GLOBALCONSTANTS DefaultPool_Numeric (* Numeric object pool constants (ID, Scale, Offset, Decimals) *)
  PACKAGE Uebungen::const::UT;
  VAR_GLOBAL CONSTANT
    InputNumber_I3 : logiBUS::utils::conversion::phys::NumericObjectPool_S := (u16ObjId := 9002, r32Scale := 0.01, i32Offset := -100000, u8Decimals := 2);
    InputNumber_I4 : logiBUS::utils::conversion::phys::NumericObjectPool_S := (u16ObjId := 9003, r32Scale := 0.01, i32Offset := -100000, u8Decimals := 2);
    OutputNumber_N3 : logiBUS::utils::conversion::phys::NumericObjectPool_S := (u16ObjId := 12002, r32Scale := 0.01, i32Offset := -100000, u8Decimals := 2);
  END_VAR
END_GLOBALCONSTANTS
